// TIA Portal V17 export
// export: Created 2025-03-07T09:17:08.3414209Z, ExportSetting WithDefaults, DisplayName Totally Integrated Automation Portal, DisplayVersion V17 Update 8, DisplayName TIA Portal Openness, DisplayVersion V17 Update 8, DisplayName TIA Portal Version Control Interface, DisplayVersion V17, DisplayName SINAMICS Startdrive Advanced, DisplayVersion V17 SP2, DisplayName SINAMICS Startdrive G110M, G120, G120C, G120D, G120P, G115D, DisplayVersion V17 SP2, DisplayName SINAMICS Startdrive G130, G150, S120, S150, SINAMICS MV, S210, DisplayVersion V17 SP2, DisplayName STEP 7 Professional, DisplayVersion V17 Update 8, DisplayName SINUMERIK ONE STEP 7 Toolbox, DisplayVersion V17 Update 12, DisplayName SINUMERIK 840D sl STEP 7 Toolbox, DisplayVersion V17 Update 12, DisplayName STEP 7 Safety, DisplayVersion V17 Update 6, DisplayName WinCC Advanced, DisplayVersion V17 Update 8
FUNCTION "FC300_CHANNELS" : Void   // FC300, LAD
{ S7_Optimized_Access := 'FALSE' }
AUTHOR : ETXETAR
VERSION : 1.0
// stored: AutoNumber false, IsIECCheckEnabled false, SetENOAutomatically false, UDAEnableTagReadback false
BEGIN

REGION Network 1: CALL FC321 CHANNEL 1 / CALL FC121
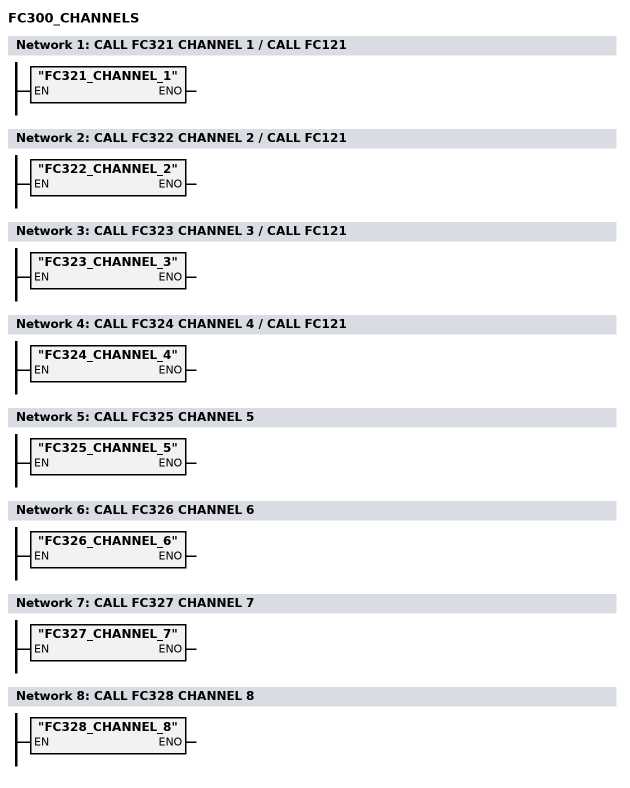
   RUNG wire#powerrail
      "FC321_CHANNEL_1"()
   END_RUNG
   // the same network as SCL:
   "FC321_CHANNEL_1"();
END_REGION

REGION Network 2: CALL FC322 CHANNEL 2 / CALL FC121
   RUNG wire#powerrail
      "FC322_CHANNEL_2"()
   END_RUNG
   // the same network as SCL:
   "FC322_CHANNEL_2"();
END_REGION

REGION Network 3: CALL FC323 CHANNEL 3 / CALL FC121
   RUNG wire#powerrail
      "FC323_CHANNEL_3"()
   END_RUNG
   // the same network as SCL:
   "FC323_CHANNEL_3"();
END_REGION

REGION Network 4: CALL FC324 CHANNEL 4 / CALL FC121
   RUNG wire#powerrail
      "FC324_CHANNEL_4"()
   END_RUNG
   // the same network as SCL:
   "FC324_CHANNEL_4"();
END_REGION

REGION Network 5: CALL FC325 CHANNEL 5
   RUNG wire#powerrail
      "FC325_CHANNEL_5"()
   END_RUNG
   // the same network as SCL:
   "FC325_CHANNEL_5"();
END_REGION

REGION Network 6: CALL FC326 CHANNEL 6
   RUNG wire#powerrail
      "FC326_CHANNEL_6"()
   END_RUNG
   // the same network as SCL:
   "FC326_CHANNEL_6"();
END_REGION

REGION Network 7: CALL FC327 CHANNEL 7
   RUNG wire#powerrail
      "FC327_CHANNEL_7"()
   END_RUNG
   // the same network as SCL:
   "FC327_CHANNEL_7"();
END_REGION

REGION Network 8: CALL FC328 CHANNEL 8
   RUNG wire#powerrail
      "FC328_CHANNEL_8"()
   END_RUNG
   // the same network as SCL:
   "FC328_CHANNEL_8"();
END_REGION
END_FUNCTION
